% RSLogix 500 project MY1ST_BAK007.RSS, saved by version 8.30.00.16 %
PROJECT "ROCKY1"    % processor: Bul.1763 MicroLogix 1100 Series B %

PROGRAM FILES
  LAD 2   3 rungs

DATA FILES
  O0 OUTPUT  4 elements
  I1 INPUT  6 elements
  S2 STATUS  66 elements
  B3 BINARY  1 elements
  T4 TIMER  1 elements
  C5 COUNTER  1 elements
  R6 CONTROL  1 elements
  N7 INTEGER  1 elements
  F8 FLOAT  1 elements

LADDER 2
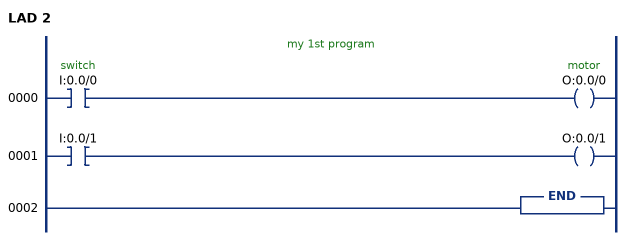
% Rung: 0 %
% my 1st program %
SOR XIC I:0.0/0 OTE O:0.0/0 EOR
%   I:0.0/0  "switch" %
%   O:0.0/0  "motor" %
% Rung: 1 %
SOR XIC I:0.0/1 OTE O:0.0/1 EOR
% Rung: 2 %
SOR END EOR
